(* PLC project Generated.project, CODESYS CODESYS V3.5 SP19 Patch 1 *)
(* stored: creationDateTime 2026-09-06T13:00:42.388378, modificationDateTime 2026-09-06T13:00:42.388378 *)

(* values of E_PresetConfirmMode: READBACK_ONLY: Confirmation par relecture de position; READBACK_AND_STATUSBIT: Relecture et bit d'état matériel; STATUSBIT_ONLY: Bit d'état matériel uniquement *)

{attribute 'qualified_only'}
{attribute 'strict'}
TYPE E_PresetConfirmMode : (READBACK_ONLY := 0, READBACK_AND_STATUSBIT := 1, STATUSBIT_ONLY := 2);
END_TYPE
